Yaskawa INFORM job: TOMASZ.JBI

/JOB
//NAME TOMASZ
//POS
///NPOS 22,22,22,3,0,0
///TOOL 0
///POSTYPE PULSE
///PULSE
C00000=-39469,-40023,29389,1619,23823,83980
C00001=-39469,-40023,29389,1619,23823,83980
C00002=-42834,34193,66784,2815,37596,82651
C00003=-4867,-51741,-21925,-16339,35132,88645
C00004=-1677,34263,22653,-17376,59387,88238
C00005=-39469,-40023,29389,1619,23823,83980
C00006=-19290,-13515,10491,-19481,22854,90941
C00007=-19594,-22569,3876,-19500,22244,90924
C00008=-44188,-83847,-61893,31337,114325,-33875
C00009=-43194,-84730,-62262,31667,113761,-33613
C00010=-44187,-83848,-61893,31338,114326,-33873
C00011=-44187,-83095,-60119,31153,113720,-34057
C00012=-44188,-83847,-61893,31337,114325,-33875
C00013=-38294,-69301,-55326,34501,114941,-31029
C00014=-37385,-70057,-55693,34765,114435,-30789
C00015=-38295,-69303,-55327,34501,114941,-31029
C00016=-38295,-68744,-53650,34283,114322,-31243
C00017=-38295,-69303,-55327,34501,114941,-31029
C00018=-46527,-81632,-60952,30529,115665,-34498
C00019=-44038,-85471,-61764,31141,113480,-34070
C00020=-37221,-68411,-54090,34763,114250,-30783
C00021=-39345,-63825,-52880,34517,116453,-30987
BC00000=135650,663732,836779
BC00001=135650,663732,836779
BC00002=135650,663662,836779
BC00003=135650,663712,836779
BC00004=186830,663711,642981
BC00005=135650,663732,836779
BC00006=136241,663732,834540
BC00007=151347,805786,834536
BC00008=353550,856982,323391
BC00009=353550,856982,323391
BC00010=353550,856982,323389
BC00011=353550,856982,323389
BC00012=353550,856982,323391
BC00013=353550,856982,323391
BC00014=353550,856982,323391
BC00015=353550,856982,323391
BC00016=353550,856982,323391
BC00017=353550,856982,323391
BC00018=353550,856982,323388
BC00019=353550,856982,323388
BC00020=353550,856982,323388
BC00021=353550,856982,323388
EC00000=4,1
EC00001=4,1
EC00002=4,-890
EC00003=4,-257
EC00004=-1211,-258
EC00005=4,1
EC00006=-10,-2
EC00007=-9,-2
EC00008=1,1
EC00009=1,1
EC00010=2,1
EC00011=2,1
EC00012=1,1
EC00013=1,1
EC00014=1,1
EC00015=1,1
EC00016=1,1
EC00017=1,1
EC00018=1,1
EC00019=1,1
EC00020=1,1
EC00021=1,1
///POSTYPE BASE
///RECTAN
///RCONF 0,0,0,0,0,0,0,0,0,0,0,0,0,0,0,0,0,0,0,0,0,0,0,0
P00006=0.222,-3.123,-1.508,0.0000,0.0000,0.0000
P00051=0.367,3.892,0.009,0.0000,0.0000,0.0000
P00052=0.088,2.832,-0.342,0.0000,0.0000,0.0000
//INST
///DATE 2024/05/16 11:48
///ATTR SC,RW
///GROUP1 RB1,BS1
///GROUP2 ST1
NOP
MOVJ C00000 BC00000 VJ=50.00  +MOVJ EC00000 VJ=100.00
MOVJ C00001 BC00001 VJ=100.00  +MOVJ EC00001 VJ=75.00
MOVJ C00002 BC00002 VJ=100.00  +MOVJ EC00002 VJ=100.00
MOVJ C00003 BC00003 VJ=75.00  +MOVJ EC00003 VJ=75.00
MOVJ C00004 BC00004 VJ=75.00  +MOVJ EC00004 VJ=75.00
MOVJ C00005 BC00005 VJ=75.00  +MOVJ EC00005 VJ=75.00
MOVL C00006 BC00006 V=500.0  +MOVJ EC00006 VJ=75.00
MOVC C00007 BC00007 V=500.0  +MOVJ EC00007 VJ=75.00
'---------------
'---------------
'---------------
SFTOF3D
SMOVL C00008 BC00008 V=100.0  +MOVJ EC00008
SREFP 3 C00009 BC00009  +REFP EC00009
CALL JOB:SEARCH-R1-S13D_TEST
SET P051 P006
SFTON3D P051
SMOVL C00010 BC00010 V=100.0  +MOVJ EC00010
SREFP 3 C00011 BC00011  +REFP EC00011
CALL JOB:SEARCH-R1-S13D_TEST
SET P051 P006
SFTON3D P051
SMOVL C00012 BC00012 V=100.0  +MOVJ EC00012
SFTOF3D
SMOVL C00013 BC00013 V=100.0  +MOVJ EC00013
SREFP 3 C00014 BC00014  +REFP EC00014
CALL JOB:SEARCH-R1-S13D_TEST
SET P052 P006
SFTON3D P052
SMOVL C00015 BC00015 V=100.0  +MOVJ EC00015
SREFP 3 C00016 BC00016  +REFP EC00016
CALL JOB:SEARCH-R1-S13D_TEST
SET P052 P006
SFTON3D P052
SFTOF3D
SMOVL C00017 BC00017 V=100.0  +MOVJ EC00017
SMOVL C00018 BC00018 V=166.7  +MOVJ EC00018
SFTON3D P051
SMOVL C00019 BC00019 V=166.7  +MOVJ EC00019
SFTON3D P052
SMOVL C00020 BC00020 V=8.3  +MOVJ EC00020
SFTOF3D
SMOVL C00021 BC00021 V=166.7  +MOVJ EC00021
END
